# EPICS autosave request: dxpApp/Db/dxpSCA_32_settings.req
$(P)$(R)NumSCAs
$(P)$(R)SCA0Low
$(P)$(R)SCA0High
$(P)$(R)SCA1Low
$(P)$(R)SCA1High
$(P)$(R)SCA2Low
$(P)$(R)SCA2High
$(P)$(R)SCA3Low
$(P)$(R)SCA3High
$(P)$(R)SCA4Low
$(P)$(R)SCA4High
$(P)$(R)SCA5Low
$(P)$(R)SCA5High
$(P)$(R)SCA6Low
$(P)$(R)SCA6High
$(P)$(R)SCA7Low
$(P)$(R)SCA7High
$(P)$(R)SCA8Low
$(P)$(R)SCA8High
$(P)$(R)SCA9Low
$(P)$(R)SCA9High
$(P)$(R)SCA10Low
$(P)$(R)SCA10High
$(P)$(R)SCA11Low
$(P)$(R)SCA11High
$(P)$(R)SCA12Low
$(P)$(R)SCA12High
$(P)$(R)SCA13Low
$(P)$(R)SCA13High
$(P)$(R)SCA14Low
$(P)$(R)SCA14High
$(P)$(R)SCA15Low
$(P)$(R)SCA15High
$(P)$(R)SCA16Low
$(P)$(R)SCA16High
$(P)$(R)SCA17Low
$(P)$(R)SCA17High
$(P)$(R)SCA18Low
$(P)$(R)SCA18High
$(P)$(R)SCA19Low
$(P)$(R)SCA19High
$(P)$(R)SCA20Low
$(P)$(R)SCA20High
$(P)$(R)SCA21Low
$(P)$(R)SCA21High
$(P)$(R)SCA22Low
$(P)$(R)SCA22High
$(P)$(R)SCA23Low
$(P)$(R)SCA23High
$(P)$(R)SCA24Low
$(P)$(R)SCA24High
$(P)$(R)SCA25Low
$(P)$(R)SCA25High
$(P)$(R)SCA26Low
$(P)$(R)SCA26High
$(P)$(R)SCA27Low
$(P)$(R)SCA27High
$(P)$(R)SCA28Low
$(P)$(R)SCA28High
$(P)$(R)SCA29Low
$(P)$(R)SCA29High
$(P)$(R)SCA30Low
$(P)$(R)SCA30High
$(P)$(R)SCA31Low
$(P)$(R)SCA31High
